Yaskawa INFORM job: 2-Y.JBI

/JOB
//NAME 2-Y
///FOLDERNAME INNE
//POS
///NPOS 2,2,0,0,0,0
///TOOL 0
///POSTYPE PULSE
///PULSE
C00000=-106078,33089,61597,-22603,72535,-32318
C00001=107766,78049,114385,24079,63734,31850
BC00000=277960,863803,688927
BC00001=277960,1283097,688929
//INST
///DATE 2023/10/04 15:13
///ATTR SC,RW
///GROUP1 RB1,BS1
NOP
MOVJ C00000 BC00000 VJ=0.78
MOVJ C00001 BC00001 VJ=0.78
END
